Staubli VAL3: Move.pgx

program Move()
begin
  //作用：运动指令运行

  //运动堆栈初始化
  resetMotion()

  //等待机械手臂上电
  wait(isPowered())

  //关节点运动
  movej(j1,tTool,mMdesc)

  //坐标点运动
  movel(p1,tTool,mMdesc)

  //等待运动指令完成
  waitEndMove()







end
